KUKA KRL program: chk_w3_wechs_ok.src

&ACCESS RV2
&REL 5
&COMMENT Check Gripper
DEF chk_w3_wechs_ok( )
Diag_Appl(#on,5)

;VERIFICAÇÃO DE FERRAMENTA: GRIPPER

$TIMER[10] = 0
$TIMER_STOP[10] = FALSE

wait for (($in[161]) and ($in[169]) and (not $in[177]) and ($in[185]) and ($in[219]))

;//---- End -------
Diag_Appl(#Off,5)

$TIMER_STOP[10] = TRUE
$TIMER[10] = 0

END
